{attribute 'qualified_only'}
{attribute 'strict'}
TYPE E_ACTUATOR_STATE :
(
	NONE	:= 0,
	NOTOP,
	OP
);
END_TYPE

(* stored: Version 1.1.0.1, ProductVersion 3.1.4024.3
   DUT E_ACTUATOR_STATE: Id {0c5e1c75-58c7-481c-a4a1-105f35a7d95f} *)
